PROGRAM MAIN
VAR
END_VAR

// Aufrufen der Objekte
Anlage();
// Aufrufen der Skills
SkillSet();
// Aufrufen der Systenparameterzuweisung 
Systemparameter();
// Aufrunfen des Zustandshandlings
Zustandshandling();
// Temporäre Punktedatenbank
PunkteZuweisung_Temp();

// Aufrufen von Testablauf
AP_V1();

END_PROGRAM

(* stored: Version 1.1.0.1
   POU MAIN: Id {312d8d08-fddc-42b7-8da4-cd7f10cc1961}, SpecialFunc None *)
